(* Schneider Machine Expert - Basic project p10, file version 1.8.0.0 *)
(* ProjectInformations: Name=New project *)

HARDWARE
  Cpu 0: TM221CE16R
  EthernetConfiguration: NetworkName=M221, IpAllocationMode=FixedAddress, IpAddress=192.168.162.202, SubnetMask=255.255.255.0
  SerialLineConfiguration: Baud=Baud19200, Parity=ParityEven, DataBits=DataBits8, StopBits=StopBits1, PhysicalMedium=PhysicalMediumRs485, TransmissionMode=TransmissionModeModbusRtu, SlaveId=1, Addressing=SlaveAddressing
  MastTask: UsePeriodScanMode=false, PeriodScan=100
  FastTask: Period=255
  CpuBehavior: StartingMode=StartAsPreviousState, AutoSaveRamOnEeprom=true, WatchdogPeriod=250

SYMBOLS  (address, symbol, comment, settings)
  %TM0        [Preset=3, Base=OneSecond, IsRetentive=true]
  %TM1        [Preset=3, Base=OneSecond, IsRetentive=true]
  %TM2        [Preset=3, Base=OneSecond, IsRetentive=true]

POU New POU
  (* SectionNumber=1 *)

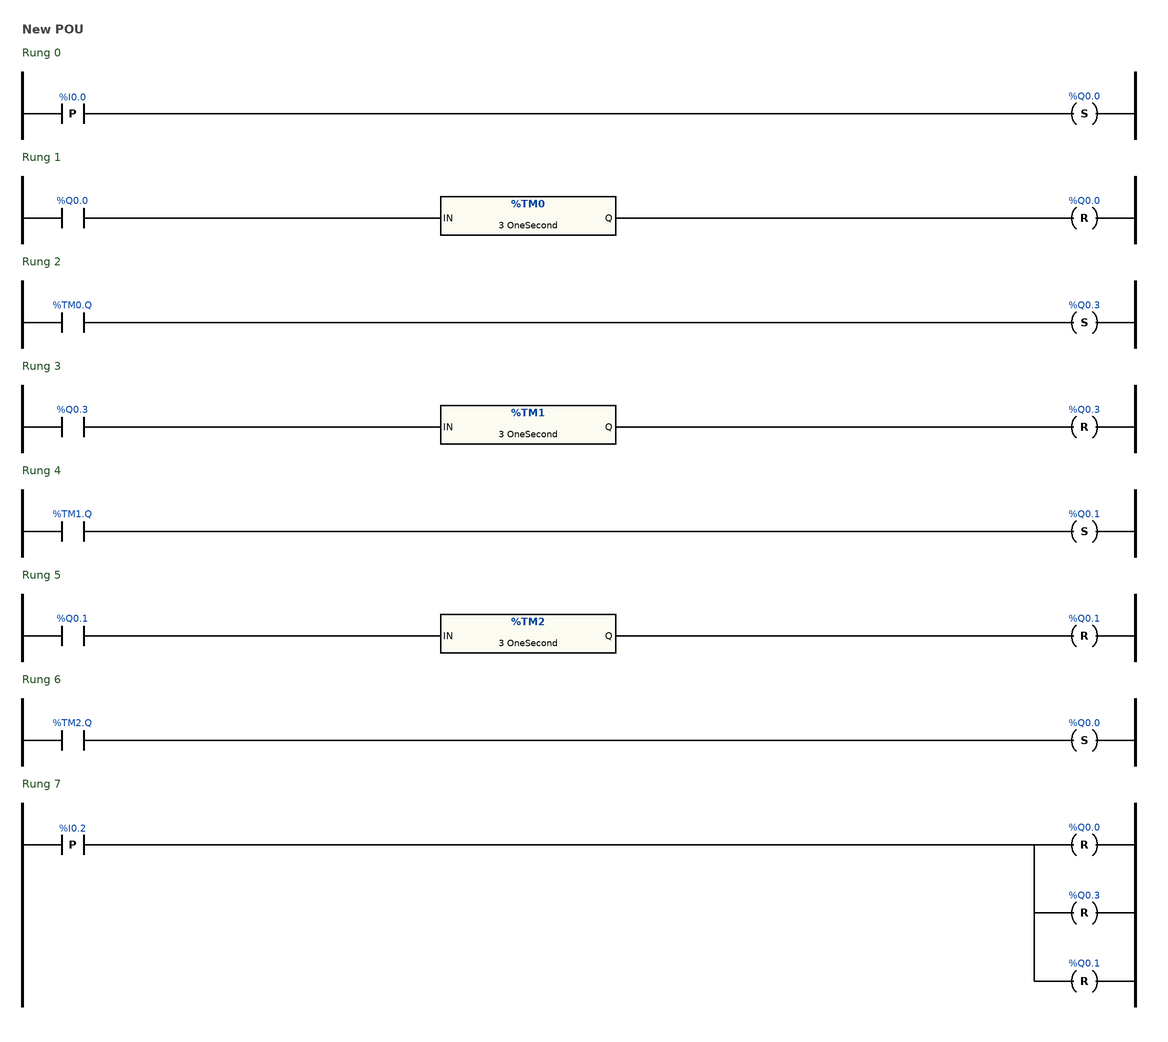

// Rung 0
  LDR %I0.0
  S %Q0.0
  // as ST:
  //   IF RISING(%I0.0) THEN %Q0.0 := TRUE; END_IF;

// Rung 1
  BLK %TM0
  LD %Q0.0
  IN
  OUT_BLK
  LD Q
  R %Q0.0
  END_BLK
  // as ST:
  //   %TM0(IN := %Q0.0);
  //   IF %TM0.Q THEN %Q0.0 := FALSE; END_IF;

// Rung 2
  LD %TM0.Q
  S %Q0.3
  // as ST:
  //   IF %TM0.Q THEN %Q0.3 := TRUE; END_IF;

// Rung 3
  BLK %TM1
  LD %Q0.3
  IN
  OUT_BLK
  LD Q
  R %Q0.3
  END_BLK
  // as ST:
  //   %TM1(IN := %Q0.3);
  //   IF %TM1.Q THEN %Q0.3 := FALSE; END_IF;

// Rung 4
  LD %TM1.Q
  S %Q0.1
  // as ST:
  //   IF %TM1.Q THEN %Q0.1 := TRUE; END_IF;

// Rung 5
  BLK %TM2
  LD %Q0.1
  IN
  OUT_BLK
  LD Q
  R %Q0.1
  END_BLK
  // as ST:
  //   %TM2(IN := %Q0.1);
  //   IF %TM2.Q THEN %Q0.1 := FALSE; END_IF;

// Rung 6
  LD %TM2.Q
  S %Q0.0
  // as ST:
  //   IF %TM2.Q THEN %Q0.0 := TRUE; END_IF;

// Rung 7
  LDR %I0.2
  R %Q0.0
  R %Q0.3
  R %Q0.1
  // as ST:
  //   IF RISING(%I0.2) THEN %Q0.0 := FALSE; END_IF;
  //   IF RISING(%I0.2) THEN %Q0.3 := FALSE; END_IF;
  //   IF RISING(%I0.2) THEN %Q0.1 := FALSE; END_IF;
